RoboDK station: AROB_S4_A6.rdk

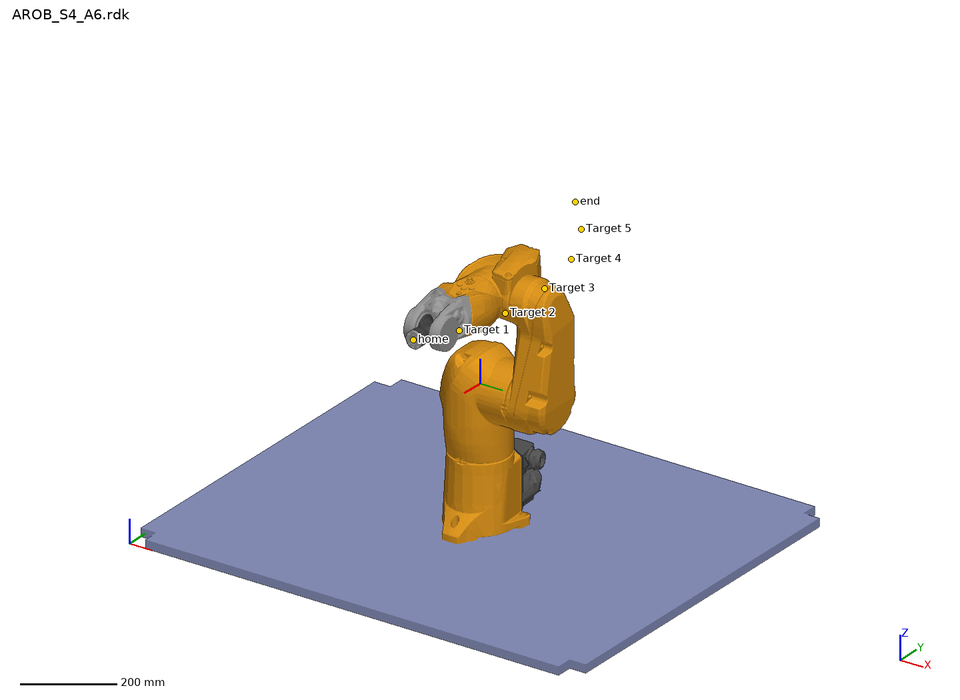
[picture v0: the station drawn from its stored meshes, robots at their saved joint values, targets as dots, program paths as lines]
Station AROB_S4_A4 (saved by RoboDK 5.6.9). Poses are relative to the parent item; angles as X-Y-Z fixed-axis rotations.
  - frame world at (0, 0, 0) mm
    - frame Staubli TX2-40 Base at (560, 460, 340) mm, rotated rx 0 ry 0 rz -90 deg
      - robot Staubli TX2-40: 6 axes, payload 2 kg, reach 515 mm, repeatability 0.02 mm, weight 29 kg
          modified DH rows (alpha deg, a mm, theta deg, d mm): 0, 0, 0, 320; -90, 0, -90, 35; 0, 225, -90, 0; -90, 0, 0, 225; 90, 0, 0, 0; -90, 0, 180, 65
          base shift (0, 0, -320) mm
          joint limits [-180, -125, -138, -270, -120, -270] to [180, 125, 138, 270, 133.5, 270]; home [0, 0, 90, 0, 0, 0]; saved at [0, 0, 90, 0, 0, 0]
    - object Arbeitsflaeche_geteilt at (0, 0, 0) mm, size 1120 x 920 x 20 mm, geometry from Arbeitsflaeche_geteilt.iges
    - object Arbeitsflaeche_komplett at (0, 0, 0) mm, size 1120 x 920 x 20 mm, geometry from Arbeitsflaeche_komplett.IGS
    - object Zelle at (0, 0, 0) mm, rotated rx 90 ry 0 rz -90 deg, size 1120 x 1947.8 x 1200 mm, geometry from Zelle.stp
    - target home (joint target) at (595, 170, 565) mm, rotated rx 0 ry 90 rz -90 deg; joints [0, 0, 90, 0, 0, 0] of Staubli TX2-40
    - target end (joint target) at (730.33, 559.49, 764.49) mm, rotated rx 62.55 ry 25.09 rz 78.25 deg; joints [118, 0, 40, -50, 33, 95] of Staubli TX2-40
    - target Target 1 (joint target) at (688.88, 200.71, 600.89) mm, rotated rx 69.05 ry 81.89 rz -1.89 deg; joints [19.667, 0, 81.667, -8.333, 5.5, 15.833] of Staubli TX2-40
    - target Target 2 (joint target) at (761.84, 263.3, 636.45) mm, rotated rx 68.33 ry 73.25 rz 15.35 deg; joints [39.333, 0, 73.333, -16.667, 11, 31.667] of Staubli TX2-40
    - target Target 3 (joint target) at (803.28, 345.55, 671.26) mm, rotated rx 67.27 ry 63.58 rz 31.44 deg; joints [59, 0, 65, -25, 16.5, 47.5] of Staubli TX2-40
    - target Target 4 (joint target) at (808.9, 432.16, 704.76) mm, rotated rx 65.97 ry 52.48 rz 46.92 deg; joints [78.667, 0, 56.667, -33.333, 22, 63.333] of Staubli TX2-40
    - target Target 5 (joint target) at (781.49, 507.65, 736.16) mm, rotated rx 64.44 ry 39.68 rz 62.36 deg; joints [98.333, 0, 48.333, -41.667, 27.5, 79.167] of Staubli TX2-40
  - Python program Prog_viaTarget (listed below)
  - Python program Prog_Direct (listed below)

--- Python program Prog_viaTarget ---
# Type help("robodk.robolink") or help("robodk.robomath") for more information
# Press F5 to run the script
# Documentation: https://robodk.com/doc/en/RoboDK-API.html
# Reference:     https://robodk.com/doc/en/PythonAPI/robodk.html
# Note: It is not required to keep a copy of this file, your Python script is saved with your RDK project
import robodk.robolink as rl    # Robot link toolbox
import time

# Link to RoboDK
RDK = rl.Robolink()

robot = RDK.Item('Staubli TX2-40')

world = RDK.Item('world')
home = RDK.Item('home')
target1 = RDK.Item('Target 1')
target2 = RDK.Item('Target 2')
target3 = RDK.Item('Target 3')
target4 = RDK.Item('Target 4')
target5 = RDK.Item('Target 5')
end = RDK.Item('end')

print('start')

robot.setAccelerationJoints(150)
robot.setSpeedJoints(75)

robot.MoveJ(home)
robot.MoveJ(target1)
robot.MoveJ(target2)
robot.MoveJ(target3)
robot.MoveJ(target4)
robot.MoveJ(target5)
robot.MoveJ(end)
time.sleep(0.1)
robot.MoveJ(target5)
robot.MoveJ(target4)
robot.MoveJ(target3)
robot.MoveJ(target2)
robot.MoveJ(target1)
robot.MoveJ(home)
print('end')

--- Python program Prog_Direct ---
# Type help("robodk.robolink") or help("robodk.robomath") for more information
# Press F5 to run the script
# Documentation: https://robodk.com/doc/en/RoboDK-API.html
# Reference:     https://robodk.com/doc/en/PythonAPI/robodk.html
# Note: It is not required to keep a copy of this file, your Python script is saved with your RDK project
import robodk.robolink as rl    # Robot link toolbox
import time
import numpy as np

# Link to RoboDK
RDK = rl.Robolink()

robot = RDK.Item('Staubli TX2-40')
world = RDK.Item('world')
home = RDK.Item('home')
target1 = RDK.Item('Target 1')
target2 = RDK.Item('Target 2')
target3 = RDK.Item('Target 3')
target4 = RDK.Item('Target 4')
target5 = RDK.Item('Target 5')
end = RDK.Item('end')

print(target1)

print('start')

robot.setAccelerationJoints(150)
robot.setSpeedJoints(75)

robot.MoveJ(home)
robot.MoveJ(end)

time.sleep(0.1)

robot.MoveJ(home)
print('end')
